GLOBALCONSTANTS quarterconst (* Global constants *)
  (* Standard: 61499-1 *)
  (* Version 1.0, 2024-02-22, franz *)
  VAR_GLOBAL CONSTANT
    BYTE_QUARTER_ZZ : BYTE := 2#0000_0000; (* ZERO Constant *)
    SHFT_QUARTER_00 : SINT := 0; (* shift 0 bits *)
    BYTE_QUARTER_00 : BYTE := 2#0000_0011; (* quarter byte 00 Constant *)
    SHFT_QUARTER_01 : SINT := 2; (* shift 2 bits *)
    BYTE_QUARTER_01 : BYTE := 2#0000_1100; (* quarter byte 01 Constant *)
    SHFT_QUARTER_02 : SINT := 4; (* shift 4 bits *)
    BYTE_QUARTER_02 : BYTE := 2#0011_0000; (* quarter byte 02 Constant *)
    SHFT_QUARTER_03 : SINT := 6; (* shift 6 bits *)
    BYTE_QUARTER_03 : BYTE := 2#1100_0000; (* quarter byte 03 Constant *)
  END_VAR
END_GLOBALCONSTANTS
